// TwinCAT 3 PLC project SafetyLogic
// ProgramVersion: 3.1.4022.1
// libraries:
//   Tc2_Standard, * (Beckhoff Automation GmbH)
//   Tc2_System, * (Beckhoff Automation GmbH)
//   Tc3_Module, * (Beckhoff Automation GmbH)
// project tree:
//   GVLs/ GVL_IO_SAFETY.TcGVL
//   POUs/ MAIN.TcPOU
//   / SafetyTask.TcTTO
// (motion and I/O tree: see PLC project plc)
// real-time tasks:
//   TASK PlcTask: cycle T#10ms, priority 20, ADS port 350
//   TASK VISU_TASK: cycle T#100000us, priority 30, ADS port 351
//   TASK SafetyTask: cycle T#10ms, priority 21, ADS port 352
//   TASK Recepty: cycle T#50000us, priority 1, ADS port 353
// variable links:
//   PLC/PLC Instance <-> SafetyLogic/SafetyLogic Instance
//     PlcTask Inputs/GVL_SafetyFrom_RT2.bSAFETY_Error <-> SafetyTask Outputs/GVL_IO_SAFETY.bSAFETY_Error
//     PlcTask Inputs/GVL_SafetyFrom_RT2.bSAFETY_FalownikKierPermitionOutSS1 <-> SafetyTask Outputs/GVL_IO_SAFETY.bSAFETY_FalownikKierPermitionOutSS1
//     PlcTask Inputs/GVL_SafetyFrom_RT2.bSAFETY_PermissionSS1 <-> SafetyTask Outputs/GVL_IO_SAFETY.bSAFETY_PermissionOutSS1
//     PlcTask Inputs/GVL_SafetyFrom_RT2.bSAFETY_PermissionSS2 <-> SafetyTask Outputs/GVL_IO_SAFETY.bSAFETY_PermissionOutSS2
//     PlcTask Inputs/GVL_SafetyFrom_RT2.bSAFETY_ResetBusy <-> SafetyTask Outputs/GVL_IO_SAFETY.bSAFETY_ResetBusy
//     PlcTask Inputs/GVL_SafetyFrom_RT2.bSAFETY_ServoKierPermitionOutSS1 <-> SafetyTask Outputs/GVL_IO_SAFETY.bSAFETY_ServoKierPermitionOutSS1
//     PlcTask Inputs/GVL_SafetyFrom_RT2.bSAFETY_ZaklejarkaKierPermitionOutSS1 <-> SafetyTask Outputs/GVL_IO_SAFETY.bSAFETY_ZaklejarkaKierPermitionOutSS1
//     PlcTask Inputs/GVL_SafetyFrom_RT2.dwGroupErrors <-> SafetyTask Outputs/GVL_IO_SAFETY.dwGroupErrors
//     PlcTask Outputs/GVL_SafetyFrom_RT2.bSAFETY_ResetCMD <-> SafetyTask Inputs/GVL_IO_SAFETY.bSAFETY_ResetCMD
//   SafetyLogic/SafetyLogic Instance <-> Device 3 (EtherCAT)/Term 1 (EK1100)/Term 2 (EL6910)
//     SafetyTask Inputs/GVL_IO_SAFETY.bCOM_ERR_TSG1 <-> StandardInputs/Standard Out Var 34
//     SafetyTask Inputs/GVL_IO_SAFETY.bCOM_ERR_TSG2 <-> StandardInputs/Standard Out Var 44
//     SafetyTask Inputs/GVL_IO_SAFETY.bFB_ERR_TSG1 <-> StandardInputs/Standard Out Var 31
//     SafetyTask Inputs/GVL_IO_SAFETY.bFB_ERR_TSG2 <-> StandardInputs/Standard Out Var 45
//     SafetyTask Inputs/GVL_IO_SAFETY.bFalownikKierownicaEStop <-> StandardInputs/Standard Out Var 71
//     SafetyTask Inputs/GVL_IO_SAFETY.bOTHER_ERR_TSG1 <-> StandardInputs/Standard Out Var 37
//     SafetyTask Inputs/GVL_IO_SAFETY.bOTHER_ERR_TSG2 <-> StandardInputs/Standard Out Var 46
//     SafetyTask Inputs/GVL_IO_SAFETY.bSafeStopAX5000 <-> StandardInputs/Standard Out Var 56
//     SafetyTask Inputs/GVL_IO_SAFETY.bSafeStopOmron <-> StandardInputs/Standard Out Var 55
//     SafetyTask Inputs/GVL_IO_SAFETY.bServoKierownicaEStop <-> StandardInputs/Standard Out Var 70
//     SafetyTask Inputs/GVL_IO_SAFETY.bZaklejarkaEStop <-> StandardInputs/Standard Out Var 72
//     SafetyTask Outputs/GVL_IO_SAFETY.bERR_ACK_TSG1 <-> StandardOutputs/Standard In Var 28
//     SafetyTask Outputs/GVL_IO_SAFETY.bERR_ACK_TSG2 <-> StandardOutputs/Standard In Var 42
//     SafetyTask Outputs/GVL_IO_SAFETY.bRUN_STOP_TSG1 <-> StandardOutputs/Standard In Var 25
//     SafetyTask Outputs/GVL_IO_SAFETY.bRUN_STOP_TSG2 <-> StandardOutputs/Standard In Var 43
//     SafetyTask Outputs/GVL_IO_SAFETY.bRestartFBs_TSG1 <-> StandardOutputs/Standard In Var 54

CONFIGURATION SafetyLogic
    RESOURCE PLC ON TwinCAT3
        TASK SafetyTask(INTERVAL := T#10ms, PRIORITY := 21);
        PROGRAM MAIN WITH SafetyTask : MAIN;
    END_RESOURCE
END_CONFIGURATION

// ---- GVLs/GVL_IO_SAFETY.TcGVL
{attribute 'qualified_only'}
VAR_GLOBAL
// ==============================================
// ======= Safety Group - inputs/outputs ========
	bFB_ERR_TSG1 				AT %I*	: BOOL;
	bCOM_ERR_TSG1 				AT %I*	: BOOL;	
	bOTHER_ERR_TSG1 			AT %I*	: BOOL;					// EL6910
	bRUN_STOP_TSG1 				AT %Q*	: BOOL 		:= TRUE;
	bERR_ACK_TSG1 				AT %Q*	: BOOL;

	bFB_ERR_TSG2 				AT %I*	: BOOL;
	bCOM_ERR_TSG2 				AT %I*	: BOOL;	
	bOTHER_ERR_TSG2 			AT %I*	: BOOL;					// EL6910
	bRUN_STOP_TSG2 				AT %Q*	: BOOL 		:= TRUE;
	bERR_ACK_TSG2 				AT %Q*	: BOOL;

	
	
	bRestartFBs_TSG1			AT %Q*	: BOOL; 				// Restart FB w grupie 1
	
	bSafeStopOmron				AT%I*	: BOOL;
	bSafeStopAX5000				AT%I*	: BOOL;
	bSafeStopKierownicatoPLC	AT%I*	: BOOL;
// ======== Communication with second RT ========
	bSAFETY_Error				AT %Q*	: BOOL;
	bSAFETY_ResetCMD 			AT %I*	: BOOL;
	bSAFETY_ResetBusy			AT %Q*	: BOOL;
	bSAFETY_PermissionOutSS1	AT %Q*	: BOOL; 				// Sygnal NC - TRUE - pozwolenie na prace
	bSAFETY_PermissionOutSS2	AT %Q*	: BOOL; 				// Sygnal NC - TRUE - pozwolenie na prace
	bSAFETY_ServoKierPermitionOutSS1		AT%Q* 	: BOOL;
	bSAFETY_FalownikKierPermitionOutSS1		AT%Q* 	: BOOL;
	bSAFETY_ZaklejarkaKierPermitionOutSS1	AT%Q* 	: BOOL;

// ======== Error and states collection =========
	dwGroupErrors				AT %Q*	: DWORD;				// Group Error collection - Communication, FB, Other...

	bServoKierownicaEStop		AT%I* 	: BOOL;
	bFalownikKierownicaEStop	AT%I* 	: BOOL;
	bZaklejarkaEStop			AT%I* 	: BOOL;

END_VAR

// ---- POUs/MAIN.TcPOU
PROGRAM MAIN
VAR
	bReset						: BOOL;
	iStep						: INT;
	tonDelay					: TON;
	bDelayReq					: BOOL;
	rtReset						: R_TRIG;	// Rising edge detection
END_VAR

GVL_IO_SAFETY.dwGroupErrors.0			:=	GVL_IO_SAFETY.bCOM_ERR_TSG1;
GVL_IO_SAFETY.dwGroupErrors.1			:=	GVL_IO_SAFETY.bFB_ERR_TSG1;
GVL_IO_SAFETY.dwGroupErrors.2			:=	GVL_IO_SAFETY.bOTHER_ERR_TSG1;
GVL_IO_SAFETY.dwGroupErrors.3			:=	GVL_IO_SAFETY.bCOM_ERR_TSG2;
GVL_IO_SAFETY.dwGroupErrors.4			:=	GVL_IO_SAFETY.bFB_ERR_TSG2;
GVL_IO_SAFETY.dwGroupErrors.5			:=	GVL_IO_SAFETY.bOTHER_ERR_TSG2;

// Error collection
GVL_IO_SAFETY.bSAFETY_Error 			:= 	(GVL_IO_SAFETY.dwGroupErrors <> 0);
// Pass signals to first RT
GVL_IO_SAFETY.bSAFETY_PermissionOutSS1 				:= GVL_IO_SAFETY.bSafeStopAX5000;
GVL_IO_SAFETY.bSAFETY_PermissionOutSS2 				:= GVL_IO_SAFETY.bSafeStopOmron;
GVL_IO_SAFETY.bSAFETY_ServoKierPermitionOutSS1	 	:= GVL_IO_SAFETY.bServoKierownicaEStop;
GVL_IO_SAFETY.bSAFETY_FalownikKierPermitionOutSS1 	:= GVL_IO_SAFETY.bFalownikKierownicaEStop;
GVL_IO_SAFETY.bSAFETY_ZaklejarkaKierPermitionOutSS1	:= GVL_IO_SAFETY.bZaklejarkaEStop;
// Reset procedure
rtReset(CLK:=GVL_IO_SAFETY.bSAFETY_ResetCMD , Q=> );
// Delay
tonDelay(PT:= T#5S);
// Procedure
CASE iStep OF
	
	0:
		IF rtReset.Q THEN
			iStep 						:= iStep + 10;
			GVL_IO_SAFETY.bSAFETY_ResetBusy := TRUE;
		END_IF
	
	10:	// Reset bledu grupy - jesli jest
		GVL_IO_SAFETY.bERR_ACK_TSG1		:= GVL_IO_SAFETY.bCOM_ERR_TSG1 OR GVL_IO_SAFETY.bFB_ERR_TSG1 OR GVL_IO_SAFETY.bOTHER_ERR_TSG1;
		GVL_IO_SAFETY.bERR_ACK_TSG2		:= GVL_IO_SAFETY.bCOM_ERR_TSG2 OR GVL_IO_SAFETY.bFB_ERR_TSG2 OR GVL_IO_SAFETY.bOTHER_ERR_TSG2;
		bDelayReq 						S= GVL_IO_SAFETY.bERR_ACK_TSG1 OR GVL_IO_SAFETY.bERR_ACK_TSG2;
		IF NOT GVL_IO_SAFETY.bERR_ACK_TSG1 AND NOT GVL_IO_SAFETY.bERR_ACK_TSG2 THEN
			IF bDelayReq THEN
				iStep 					:= iStep + 5;
			ELSE
				iStep 					:= iStep + 10;
			END_IF
		END_IF	
	15: // Delay
		tonDelay.IN 					:= TRUE;
		IF tonDelay.Q THEN
			bDelayReq	 				:= FALSE;
			tonDelay.IN 				:= FALSE;
			iStep 						:= iStep + 5;
		END_IF
	20:
		GVL_IO_SAFETY.bRestartFBs_TSG1	:= TRUE;
		iStep 							:= iStep + 10;

	30:
		GVL_IO_SAFETY.bRestartFBs_TSG1	:= FALSE;
		iStep 							:= iStep + 10;	
	40:			
		GVL_IO_SAFETY.bSAFETY_ResetBusy := FALSE;				
		iStep := 0;
END_CASE

END_PROGRAM
